PROGRAM multiControl
VAR
	multiCtrlFrameIndex : INT; //Index used to switch frame on multiControlScreen
	
	aActionList : ARRAY[1..4] OF STRING := ['BMW','FORD','MERCEDES','FIAT'];
	pMotorRef1 : POINTER TO FB_teknicMotorEC;
	pMotorRef2 : POINTER TO FB_teknicMotorEC;
	pMotorRef3 : POINTER TO FB_teknicMotorEC;
	pMotorRef4 : POINTER TO FB_teknicMotorEC;
	aMotorRef :ARRAY[1..4] OF POINTER TO FB_teknicMotorEC;


	// Motor Disp //
	nMotorControlIndex : INT; // Index used to change disp of motor controls. 0-Rotation, 1- Clamping, 2-Columns, 3-Width. 
	bMotorEnable1 : BOOL;
	bMotorEnable2 : BOOL;
	bMotorEnable3 : BOOL;
	bMotorEnable4 : BOOL;

	bHideDispMotor3 : BOOL; //Used to hide or show controls for motor 3. 
	bHideDispMotor4	: BOOL;
	
	sMotorDisp1 : STRING; // Used to dynamically change the title of motor 1. 
	sMotorDisp2 : STRING;
	sMotorDisp3 : STRING;
	sMotorDisp4 : STRING;
	
	nCounter : INT;
	aMotorSpeed : ARRAY[1..4] OF LREAL;
	aMotorPos : ARRAY[1..4] OF LREAL;
	aMotorTorque : ARRAY[1..4] OF LREAL;
END_VAR

CASE nMotorControlIndex OF 
	0:// Rotation Selected
		IF bMotorEnable1 THEN
			pMotorRef1 := ADR(GVL_devices.fbLftRotationMotor);
		ELSE
			pMotorRef1 := 0;
		END_IF
		IF bMotorEnable2 THEN
			pMotorRef2 := ADR(GVL_devices.fbRhtRotationMotor);
		ELSE
			pMotorRef2 := 0;
		END_IF
		pMotorRef3 := 0;
		pMotorRef4 := 0;
	    bHideDispMotor3 := TRUE;
	    bHideDispMotor4 := TRUE;
		sMotorDisp1 := 'LEFT ROTATION';
		sMotorDisp2 := 'RIGHT ROTATION';
		sMotorDisp3 := '';
		sMotorDisp4 := '';
	1:// Clamping Selected
		IF bMotorEnable1 THEN
			pMotorRef1 := ADR(GVL_devices.fbLftClampMotor);
		ELSE
			pMotorRef1 := 0;
		END_IF
		IF bMotorEnable2 THEN
			pMotorRef2 := ADR(GVL_devices.fbRhtClampMotor);
		ELSE
			pMotorRef2 := 0;
		END_IF
		pMotorRef3 := 0;
		pMotorRef4 := 0;
	    bHideDispMotor3 := TRUE;
	    bHideDispMotor4 := TRUE;
		sMotorDisp1 := 'LEFT CLAMPING';
		sMotorDisp2 := 'RIGHT CLAMPING';
		sMotorDisp3 := '';
		sMotorDisp4 := '';
	2:// Columns Selected
		IF bMotorEnable1 THEN
			pMotorRef1 := ADR(GVL_devices.fbColumn0Motor);
		ELSE
			pMotorRef1 := 0;
		END_IF
		IF bMotorEnable2 THEN
			pMotorRef2 := ADR(GVL_devices.fbColumn1Motor);
		ELSE
			pMotorRef2 := 0;
		END_IF
		IF bMotorEnable3 THEN
			pMotorRef3 := ADR(GVL_devices.fbColumn2Motor);
		ELSE
			pMotorRef3 := 0;
		END_IF
		IF bMotorEnable4 THEN
			pMotorRef4 := ADR(GVL_devices.fbColumn3Motor);
		ELSE
			pMotorRef4 := 0;
		END_IF
	    bHideDispMotor3 := FALSE;
	    bHideDispMotor4 := FALSE;
		sMotorDisp1 := 'COLUMN 0';
		sMotorDisp2 := 'COLUMN 1';
		sMotorDisp3 := 'COLUMN 2';
		sMotorDisp4 := 'COLUMN 3';
	3:// Width Selected
		IF bMotorEnable1 THEN
			pMotorRef1 := ADR(GVL_devices.fbLftWidthMotor);
		ELSE
			pMotorRef1 := 0;
		END_IF
		IF bMotorEnable2 THEN
			pMotorRef2 := ADR(GVL_devices.fbRhtWidthMotor);
		ELSE
			pMotorRef2 := 0;
		END_IF
		pMotorRef3 := 0;
		pMotorRef4 := 0;
	    bHideDispMotor3 := TRUE;
	    bHideDispMotor4 := TRUE;
		sMotorDisp1 := 'LEFT WIDTH';
		sMotorDisp2 := 'RIGHT WIDTH';
		sMotorDisp3 := '';
		sMotorDisp4 := '';
END_CASE

aMotorRef[1] := pMotorRef1;
aMotorRef[2] := pMotorRef2;
aMotorRef[3] := pMotorRef3;
aMotorRef[4] := pMotorRef4;

FOR nCounter := 1 TO 4 BY 1 DO
	IF aMotorRef[nCounter] <> 0 THEN
		aMotorSpeed[nCounter] := aMotorRef[nCounter]^.fbMotor.NcToPlc.ActVelo;
	END_IF
END_FOR

FOR nCounter := 1 TO 4 BY 1 DO
	IF aMotorRef[nCounter] <> 0 THEN
		aMotorPos[nCounter] := aMotorRef[nCounter]^.fbMotor.NcToPlc.ActPos;
	END_IF
END_FOR

FOR nCounter := 1 TO 4 BY 1 DO
	IF aMotorRef[nCounter] <> 0 THEN
		aMotorTorque[nCounter] := aMotorRef[nCounter]^.fbMotor.NcToPlc.ActTorque;
	END_IF
END_FOR

END_PROGRAM

(* stored: Version 1.1.0.1, ProductVersion 3.1.4024.13
   POU multiControl: Id {7ac8876c-7553-4aa3-8d03-b92ac1cc6e8f}, SpecialFunc None *)
